FUNCTION_BLOCK E_SH (* Sample-and-Hold for BOOL *)
  (* Standard: 61499-2; Description: Copyright (c) 2024 HR Agrartechnik GmbH This program and the accompanying materials are made available under the terms of the Eclipse Public License 2.0 which is available at https://www.eclipse.org/legal/epl-2.0/ SPDX-License-Identifier: EPL-2.0 *)
  (* Version 1.0, 2024-02-23, franz *)
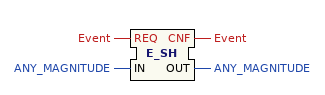
  EVENT_INPUT
    REQ; (* Normal Execution Request *)
  END_EVENT
  EVENT_OUTPUT
    CNF; (* Execution Confirmation *)
  END_EVENT
  VAR_INPUT
    IN : ANY_MAGNITUDE; (* Sample *)
  END_VAR
  VAR_OUTPUT
    OUT : ANY_MAGNITUDE; (* Hold *)
  END_VAR
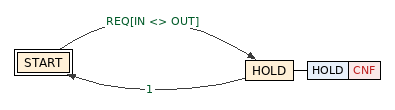
  EC_STATES
    START; (* Initial State *)
    HOLD : HOLD -> CNF;
  END_STATES
  EC_TRANSITIONS
    START TO HOLD := REQ[IN <> OUT];
    HOLD TO START := 1;
  END_TRANSITIONS
  ALGORITHM HOLD IN ST:
OUT := IN;
  END_ALGORITHM
END_FUNCTION_BLOCK
